INTERFACE ITestRunner

METHOD AddTest : BOOL
VAR_INPUT
    UnitTest : IUnitTest;
END_VAR
END_METHOD

END_INTERFACE

(* stored: Version 1.1.0.1, ProductVersion 3.1.4024.4
   Itf ITestRunner: Id {f50247c5-3d93-47fa-b020-c410187201dd}
   Method AddTest: Id {90b4c5d1-d46e-4b5e-b4b9-2103cb99f47e} *)
